FUNCTION f_calcul : REAL
VAR_INPUT
	IrAngle : REAL;
	IrHypotenuse : REAL;
END_VAR

f_calcul:=IrHypotenuse*SIN(IrAngle);

END_FUNCTION

(* stored: Version 1.1.0.1, ProductVersion 3.1.4020.6
   POU f_calcul: Id {dd262f3c-feec-4644-810a-3295bb366717}, SpecialFunc None *)
